Universal Robots PolyScope program: group.urp

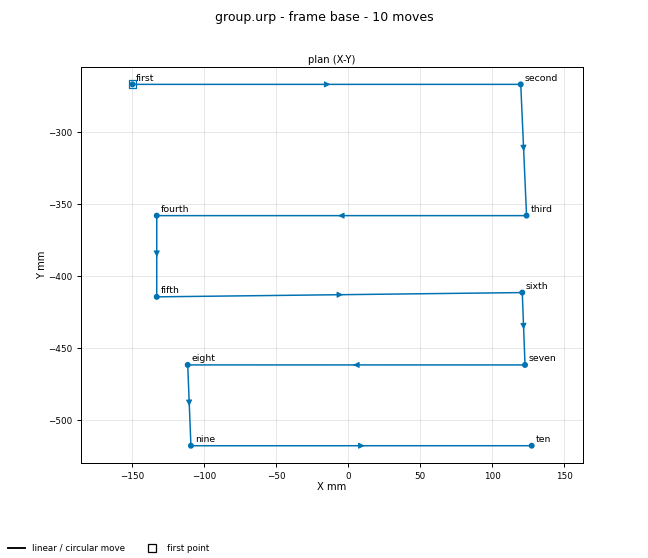
[picture p0: tool path of group.urp in frame base, 10 of 10 moves have a stored position in this frame; points joined in program order, loops and branches not executed]
Program group (installation=default directory=/programs/usbdisk_2 createdIn=5.15.2 lastSavedIn=5.15.2 robotSerialNumber=20245300417)
Calibrated DH parameters: a=[-0.000151, -0.230235, -0.197005, 0.000062, -0.000115, 0]; d=[0.151936, 15.763129, 4.882528, -20.514754, 0.085216, 0.091878]; alpha=[1.570572, -0.005074, 0.003966, 1.570169, -1.572724, 0]; deltaTheta=[0, -0.334375, 7.011453, -0.393893, 0.000003, 0]
InitVariablesNode
Robot Program (runOnlyOnce=false)
  MoveL speed 250 mm/s, acceleration 1200 mm/s^2 (useActiveTCP=true) feature=Base
    Waypoint first: TCP in base x=-149.642 y=-266.702 z=36.437 mm, rx=2.9024 ry=-1.2021 rz=0.0002 rad; joints [-95.196, -109.055, -127.577, -33.253, 90.026, -139.88] deg; TCP offset x=1.321 y=-5.838 z=76.106 mm, rx=0 ry=0 rz=0 rad
    Waypoint second: TCP in base x=119.971 y=-266.697 z=36.422 mm, rx=2.9024 ry=-1.2022 rz=0.0001 rad; joints [-40.706, -105.818, -132.903, -31.167, 90.028, -85.371] deg
    Waypoint third: TCP in base x=123.997 y=-357.852 z=36.429 mm, rx=2.9025 ry=-1.2022 rz=0.0001 rad; joints [-51.818, -121.211, -105.859, -42.815, 89.997, -96.577] deg
    Waypoint fourth: TCP in base x=-132.799 y=-357.858 z=36.432 mm, rx=2.9025 ry=-1.2021 rz=0.0002 rad; joints [-91.29, -122.339, -103.739, -43.807, 89.999, -136.058] deg
    Waypoint fifth: TCP in base x=-132.809 y=-414.252 z=36.436 mm, rx=2.9024 ry=-1.2022 rz=0.0002 rad; joints [-91.09, -132.25, -84.656, -52.979, 89.982, -135.933] deg
    Waypoint sixth: TCP in base x=121.031 y=-411.279 z=36.446 mm, rx=-2.9024 ry=1.2022 rz=-0.0003 rad; joints [-56.809, -130.445, -88.186, -51.251, 89.988, -101.637] deg
    Waypoint seven: TCP in base x=122.936 y=-461.538 z=36.46 mm, rx=2.9025 ry=-1.2021 rz=0.0004 rad; joints [-60.013, -140.719, -67.834, -61.325, 89.972, -104.93] deg
    Waypoint eight: TCP in base x=-111.299 y=-461.524 z=36.443 mm, rx=2.9025 ry=-1.2021 rz=0.0001 rad; joints [-88.289, -140.636, -68.002, -61.249, 89.97, -133.205] deg
    Waypoint nine: TCP in base x=-109.074 y=-517.644 z=36.44 mm, rx=2.9025 ry=-1.2021 rz=0.0002 rad; joints [-88.15, -156.401, -35.83, -77.656, 89.953, -133.208] deg
    Waypoint ten: TCP in base x=127.572 y=-517.631 z=36.417 mm, rx=-2.9025 ry=1.2021 rz=-0.0001 rad; joints [-62.598, -157.167, -34.246, -78.474, 89.95, -107.665] deg
